SUBAPPLICATION Uebung_080c (* Beispiel für E_CTU *)
  (* Standard: 61499-2; Description: Copyright (c) 2023 Meisterschulen am Ostbahnhof This program and the accompanying materials are made available under the terms of the Eclipse Public License 2.0 which is available at https://www.eclipse.org/legal/epl-2.0/ SPDX-License-Identifier: EPL-2.0 Beispiel für E_CTU Aufwärts zählen UAO Curriculum Module 3 - The IEC 61499 Standard, Seite 92 *)
  (* Version 1.0, 2023-10-23, Franz Höpfinger, Meisterschulen am Ostbahnhof *)
  PACKAGE Uebungen;
  IMPORT logiBUS::io::DI::logiBUS_DI::Input_I1;
  IMPORT logiBUS::io::DI::logiBUS_DI::Input_I2;
  IMPORT logiBUS::io::DI::logiBUS_DI_Events::BUTTON_SINGLE_CLICK;
  IMPORT logiBUS::io::DQ::logiBUS_DO::Output_Q1;
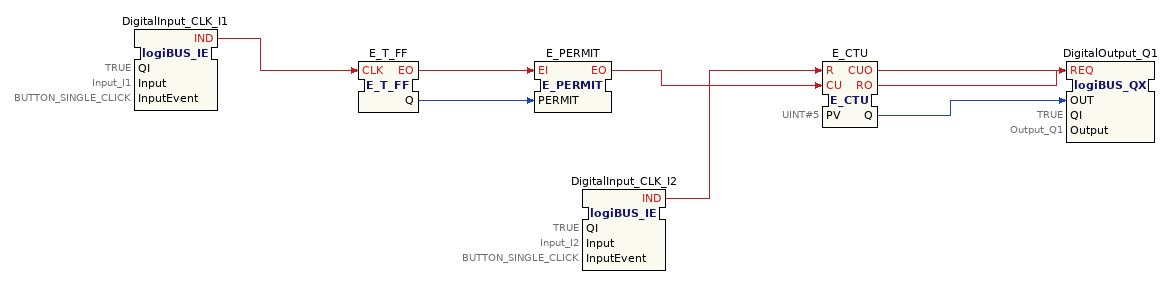
  (* Die Kombination von T_FF und PERMIT halbiert die Events. *)
  FBS
    DigitalOutput_Q1 : logiBUS::io::DQ::logiBUS_QX(QI := TRUE, Output := Output_Q1);
    DigitalInput_CLK_I1 : logiBUS::io::DI::logiBUS_IE(QI := TRUE, Input := Input_I1, InputEvent := BUTTON_SINGLE_CLICK);
    E_CTU : iec61499::events::E_CTU(PV := UINT#5);
    DigitalInput_CLK_I2 : logiBUS::io::DI::logiBUS_IE(QI := TRUE, Input := Input_I2, InputEvent := BUTTON_SINGLE_CLICK);
    E_PERMIT : iec61499::events::E_PERMIT;
    E_T_FF : iec61499::events::E_T_FF;
  END_FBS
  EVENT_CONNECTIONS
    E_CTU.CUO TO DigitalOutput_Q1.REQ;
    E_CTU.RO TO DigitalOutput_Q1.REQ;
    DigitalInput_CLK_I2.IND TO E_CTU.R;
    E_T_FF.EO TO E_PERMIT.EI;
    DigitalInput_CLK_I1.IND TO E_T_FF.CLK;
    E_PERMIT.EO TO E_CTU.CU;
  END_CONNECTIONS
  DATA_CONNECTIONS
    E_CTU.Q TO DigitalOutput_Q1.OUT;
    E_T_FF.Q TO E_PERMIT.PERMIT;
  END_CONNECTIONS
END_SUBAPPLICATION
